// TIA Portal V17 export
// export: Created 2022-05-07T16:38:48.2803166Z, ExportSetting WithDefaults, DisplayName Totally Integrated Automation Portal, DisplayVersion V17 Update 3, DisplayName TIA Portal Openness, DisplayVersion V17 Update 3, DisplayName TIA Portal Version Control Interface, DisplayVersion V17, DisplayName TIA Portal Test Suite Advanced, DisplayVersion V17 Update 1, DisplayName SINAMICS Startdrive Advanced, DisplayVersion V17 Update2, DisplayName SINAMICS Startdrive G130, G150, S120, S150, SINAMICS MV, S210, DisplayVersion V17 Update2, DisplayName SINAMICS Startdrive G110M, G120, G120C, G120D, G120P, G115D, DisplayVersion V17 Update2, DisplayName STEP 7 Professional, DisplayVersion V17 Update 3, DisplayName STEP 7 Safety, DisplayVersion V17, DisplayName WinCC UA Professional, DisplayVersion V17 Update 3
DATA_BLOCK "CTRL_ASSE_DB"   // DB4
VERSION : 0.1
// stored: AutoNumber true, DBAccessibleFromOPCUA true, InstanceOfName CTRL_ASSE_STD, InstanceOfType FB
"CTRL_ASSE_STD"
   // VAR_INPUT
   //    Automatico : Bool;
   //    Exe_MC_Reset : Bool;
   //    En_MC_Power : Bool;
   //    Exe_MC_Home : Bool;
   //    Sp_Offset_Homing : Real;
   //    Sp_Homing_Mode : Int;
   //    Exe_MC_Halt : Bool;
   //    Exe_Jog_Fwd : Bool;
   //    Exe_Jog_Bkw : Bool;
   //    Sp_Jog_Velocity : Real;
   //    Exe_MC_Velocity : Bool;
   //    Sp_MC_Velocity : Real;
   //    Exe_MC_Relative : Bool;
   //    Sp_MoveRel_Distance : Real;
   //    Sp_MoveRel_Velocity : Real;
   //    Exe_MC_Abs : Bool;
   //    Sp_MoveAbs_Position : Real;
   //    Sp_MoveAbs_Velocity : Real;
   //    Exe_MC_ChangeDyna : Bool;
   //    Sp_RampUpTime : Real;
   //    Sp_RampDnTime : Real;
   // END_VAR
   // VAR_OUTPUT
   //    Output_MC_Reset_Done : Bool;
   //    Output_MC_AxisEnabled : Bool;
   //    Output_MC_AxisHomed : Bool;
   //    Output_MC_Halt_Done : Bool;
   //    Output_MC_JogInVelocity : Bool;
   //    Output_MC_MoveInVelocity : Bool;
   //    Output_MC_MoveRel_Done : Bool;
   //    Output_MC_MoveAbs_Done : Bool;
   //    Output_MC_MoveAbs_Busy : Bool;
   //    Output_MC_At_Standstill : Bool;
   //    Output_MC_Error : Bool;
   //    Output_ActVelocity : Real;
   //    Output_ActPos : Real;
   // END_VAR
   // VAR_IN_OUT
   //    AxisTO : TO_PositioningAxis;
   // END_VAR
   // VAR
   //    AxisReady_PosAxis { S7_SetPoint := 'True'} : Bool;
   //    MC_Power_Instance { S7_SetPoint := 'True'} : MC_Power;
   //    MC_Reset_Instance { S7_SetPoint := 'True'} : MC_Reset;
   //    MC_Halt_Instance { S7_SetPoint := 'True'} : MC_Halt;
   //    MC_MoveJog_Instance { S7_SetPoint := 'True'} : MC_MoveJog;
   //    MC_MoveAbsolute_Instance { S7_SetPoint := 'True'} : MC_MoveAbsolute;
   //    MC_MoveVelocity_Instance { S7_SetPoint := 'True'} : MC_MoveVelocity;
   //    MC_Home_Instance { S7_SetPoint := 'True'} : MC_Home;
   //    MC_MoveRelative_Instance { S7_SetPoint := 'True'} : MC_MoveRelative;
   //    MC_ChangeDynamic_Instance { S7_SetPoint := 'True'} : MC_ChangeDynamic;
   // END_VAR
BEGIN
END_DATA_BLOCK
